// TIA Portal V21 export
VAR_GLOBAL   // PLC tag table "GruppoRiempiReciveDigitali"
END_VAR
VAR_GLOBAL CONSTANT   // user constants
   K_SegnaleDaGruppoRiempi_CanStopAperto : Int := 1;
END_VAR
